{attribute 'GeneratedUsingTerminal: IODEVICETYPE_ETHERCATPROT'}
{attribute addProperty BoxType "IODEVICETYPE_ETHERCATPROT"}
{attribute addProperty Id "Beckhoff_EJ1xxxBeckhoff_EJ1xxx_70A93D0A113Beckhoff_EJ2xxxBeckhoff_EJ2xxx_9E959597222Beckhoff_EJ3xxxBeckhoff_EJ3xxx_86133EA31028Beckhoff_EJ4xxxBeckhoff_EJ4xxx_1A056743105Beckhoff_EJ5xxxBeckhoff_EJ5xxx_351E5D24110Beckhoff_EJ6xxxBeckhoff_EJ6xxx_18D9AE06140Beckhoff_EJ7xxxBeckhoff_EJ7xxx_81983D091059Beckhoff_EJ9xxxBeckhoff_EJ9xxx_97F7600592Beckhoff_EJx9xxBeckhoff_EJx9xx_631E2D1F366SyncUnitsSyncUnits_99E584AF18InputsInputs_25A0042B160OutputsOutputs_2397A10E106InfoDataInfoData_C76BEFB322"}
{attribute addProperty CRC "2399612719"}
{attribute addProperty Size "3541"}
TYPE EtherCAT_Master_EJxxxx_8F072F2F :
STRUCT
	{attribute addProperty Name "Beckhoff_EJ1xxx"}
	{attribute addProperty PreviousPort "EtherCAT_Master_EJxxxx : Master"}
	Beckhoff_EJ1xxx : Beckhoff_EJ1xxx_70A93D0A;
	{attribute addProperty Name "Beckhoff_EJ2xxx"}
	{attribute addProperty PreviousPort "Beckhoff EJ1xxx : C"}
	Beckhoff_EJ2xxx : Beckhoff_EJ2xxx_9E959597;
	{attribute addProperty Name "Beckhoff_EJ3xxx"}
	{attribute addProperty PreviousPort "Beckhoff EJ2xxx : C"}
	Beckhoff_EJ3xxx : Beckhoff_EJ3xxx_86133EA3;
	{attribute addProperty Name "Beckhoff_EJ4xxx"}
	{attribute addProperty PreviousPort "Beckhoff EJ3xxx : C"}
	Beckhoff_EJ4xxx : Beckhoff_EJ4xxx_1A056743;
	{attribute addProperty Name "Beckhoff_EJ5xxx"}
	{attribute addProperty PreviousPort "Beckhoff EJ4xxx : C"}
	Beckhoff_EJ5xxx : Beckhoff_EJ5xxx_351E5D24;
	{attribute addProperty Name "Beckhoff_EJ6xxx"}
	{attribute addProperty PreviousPort "Beckhoff EJ5xxx : C"}
	Beckhoff_EJ6xxx : Beckhoff_EJ6xxx_18D9AE06;
	{attribute addProperty Name "Beckhoff_EJ7xxx"}
	{attribute addProperty PreviousPort "Beckhoff EJ6xxx : C"}
	Beckhoff_EJ7xxx : Beckhoff_EJ7xxx_81983D09;
	{attribute addProperty Name "Beckhoff_EJ9xxx"}
	{attribute addProperty PreviousPort "Beckhoff EJ7xxx : C"}
	Beckhoff_EJ9xxx : Beckhoff_EJ9xxx_97F76005;
	{attribute addProperty Name "Beckhoff_EJx9xx"}
	{attribute addProperty PreviousPort "Beckhoff EJ9xxx : C"}
	Beckhoff_EJx9xx : Beckhoff_EJx9xx_631E2D1F;
	{attribute addProperty Name "SyncUnits"}
	SyncUnits : SyncUnits_99E584AF;
	{attribute addProperty Name "Inputs"}
	Inputs : Inputs_25A0042B;
	{attribute addProperty Name "Outputs"}
	Outputs : Outputs_2397A10E;
	{attribute addProperty Name "InfoData"}
	InfoData : InfoData_C76BEFB3;
END_STRUCT
END_TYPE

(* stored: Version 1.2.0.0, ProductVersion 3.1.4024.9
   DUT EtherCAT_Master_EJxxxx_8F072F2F: Id {3e347045-f02f-4281-ace2-0e6f38bfc374} *)
